FUNCTION_BLOCK EL1084
VAR
	_io : EL1xx4_Data;
	{attribute addProperty Name "WcState"}
	_wcState : WcStateInputToggle;
	{attribute addProperty Name "Info data"}
	_infoData : InfoDataBase;
END_VAR

PROPERTY IO : REFERENCE TO EL1xx4_Data
GET
IO REF= _io;
END_GET
END_PROPERTY

PROPERTY WcState : REFERENCE TO WcStateInputToggle
GET
WcState REF= _wcState;
END_GET
END_PROPERTY

END_FUNCTION_BLOCK

(* stored: Version 1.1.0.1, ProductVersion 3.1.4024.9
   POU EL1084: Id {d13f9244-0b5c-05be-1199-e198c62bafa0}, SpecialFunc None
   Property IO: Id {29b7863c-dcdc-003a-3a2c-c4a8b356f4c3}
   Get Get: Id {d2480018-3144-0b69-1ee6-6180d90b281a}
   Property WcState: Id {ea4928d7-1cfc-0383-0f79-dc30d7c6b221}
   Get Get: Id {22d677d3-e8c7-005a-387a-afe275878b4e} *)
